Staubli VAL3: pallet_getList.pgx

program pallet_getList()
  local num i
  local num l_nSize
  local string l_sItem
begin
  // get the full pallet list, copy into sPalletName
  call pallet:getSize(l_nSize)
  if size(sPalletName)!=l_nSize
    resize(sPalletName,1,l_nSize)
  endIf
  for i=0 to l_nSize-1
    call pallet:get(l_sItem,i)
    sPalletName[i]=l_sItem
  endFor
end
